// TIA Portal V21 export
FUNCTION_BLOCK "BranchShapes"   // FB42, LAD
   VAR_TEMP   // added for the SCL form of the ladder/FBD networks
      _variant1 : Variant;
   END_VAR
BEGIN

REGION Network 1: Nested groups separated by a real contact
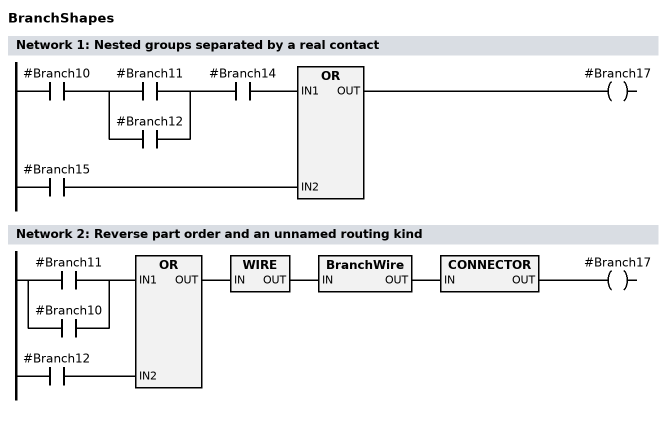
   #_variant1 := (#Branch10 AND (#Branch11 OR #Branch12) AND #Branch14) OR #Branch15;
   #Branch17 := #_variant1;
END_REGION

REGION Network 2: Reverse part order and an unnamed routing kind
   // no SCL statement known for BranchWire, Connector, Wire: written as a call
   #_variant1 := (#Branch10 OR #Branch11) OR #Branch12;
   #Branch17 := Connector(BranchWire(Wire(#_variant1)));
END_REGION
END_FUNCTION_BLOCK
